FUNCTION_BLOCK TcoContext_Waveform EXTENDS TcoCore._internals_TcoContext
VAR
	_TcoObject_Waveform		:	TcoObject_Waveform(THIS^);
END_VAR

METHOD PROTECTED  Main
_TcoObject_Waveform();
END_METHOD

END_FUNCTION_BLOCK

(* stored: Version 1.1.0.1
   POU TcoContext_Waveform: Id {76c1cbb5-02cf-02d0-2e44-70ab9bc25555}, SpecialFunc None
   Method Main: Id {229b1708-b47b-0826-0b45-44b4bc509029} *)
